FUNCTION GetSystemTimeAsTime : TIME
VAR_INPUT
END_VAR
VAR
END_VAR

GetSystemTimeAsTime := TO_TIME(F_GetSystemTime() / 10000);

END_FUNCTION

(* stored: Version 1.1.0.1, ProductVersion 3.1.4024.6
   POU GetSystemTimeAsTime: Id {7bc5a8b7-19f7-4eca-ae2b-bdf4cbf64266}, SpecialFunc None *)
